{attribute 'qualified_only'}
VAR_GLOBAL PERSISTENT
		// wejścia cyfrowe
	user_array 					: ARRAY[1..100] OF ST_UserManagment;  // Tablica użytkowników
    currentUser 				: INT := 1;  // Indeks bieżącego użytkownika (zaczyna od 1)
    string_of_properties 		: STRING(1000);  // String z HMI z danymi użytkowników
	outside_accept_login		:BOOL;
	outside_login_pool			:STRING(255);  
	new_user_added				:BOOL;		//dodano użytkownika w PLC
	user_eddited				:BOOL; 		//zedytowano użytkownika w PLC
	b_new_users					:BOOL;		//wgranie uzytkowników
	currentUserName 			:WSTRING(255);
	currentUserGroup			:STRING(80);
	actualUserOn_UserName		:STRING(80);
	b_rewrite_main_users		:BOOL:=FALSE;
	
	logout						:BOOL;
	
	user_try_to_log				:BOOL;
	user_accept_to_log_in		:BOOL;
	no_user_found				:BOOL;
	user_succesed_log			:BOOL;
	putted_user_password		:STRING(255);  //pole w które użytkownik wpisuje hasło
	
	new_user					:BOOL;			//inicjalizacja dodawania nowego użytkownika
	new_user_accept				:BOOL;			//akceptacja dodania nowego użytkownika
	newuserNameSurname 			:WSTRING(255);	//imię i nazwisko
	newpassword					:STRING(255);	//hasło
	newpasswordRFID				:STRING(255);	//hasło rfid
	newpasswordQR				:STRING(255);	//hasło qr
	newuserGroup				:STRING(80);		//grupa użytkowników
	newautoLogOff				:STRING(80);			//czas do wylogowania
	newlocale					:STRING(80);		//gdzie zapisujemy
	newtimeFormatlocale			:STRING(80);		//format godziny
	newtimeZone					:STRING(80);		//strefa czasowa
	
	edit_user					:BOOL;				//inicjalizacja edycji użytkownika
	edit_user_accept			:BOOL;			//akceptacja edycji użytkownika
	actual_editted_user			:WSTRING(255);	//wybór aktualnie edytowanego użytkownika
	edituserNameSurname 		:WSTRING(255);	//imię i nazwisko
	editpassword				:STRING(255);	//hasło
	editpasswordRFID			:STRING(255);	//hasło rfid
	editpasswordQR				:STRING(255);	//hasło qr
	edituserGroup				:STRING(80);		//grupa użytkowników
	editautoLogOff				:STRING(80);			//czas do wylogowania
	edit_user_qr_or_rfid_password	:BOOL;		//edycja kodów rfid lub qr
		
	//wyjścia cyfrowe
	new_user_add_error			:BOOL;
	edit_user_error				:BOOL;
	bwait						:BOOL;
		
	delete_user						:BOOL;
	delete_user_accept				:BOOL;
	delete_user_error				:BOOL;
	choosen_to_delete				:WSTRING(255);
	user_deleted_succes				:BOOL;
	
	password_to_log_in				:STRING(80); //hasło do pola (1 z 5 (adm, opr, ser, tech, mech)
	
	b_rewrite_users_after_issues	:BOOL:=FALSE;
	
	
END_VAR

(* stored: Version 1.1.0.1, ProductVersion 3.1.4024.12
   GVL GVL_USER_UP: Id {4fa063b0-7f01-4c6d-8d35-72eeb8a8484c} *)
